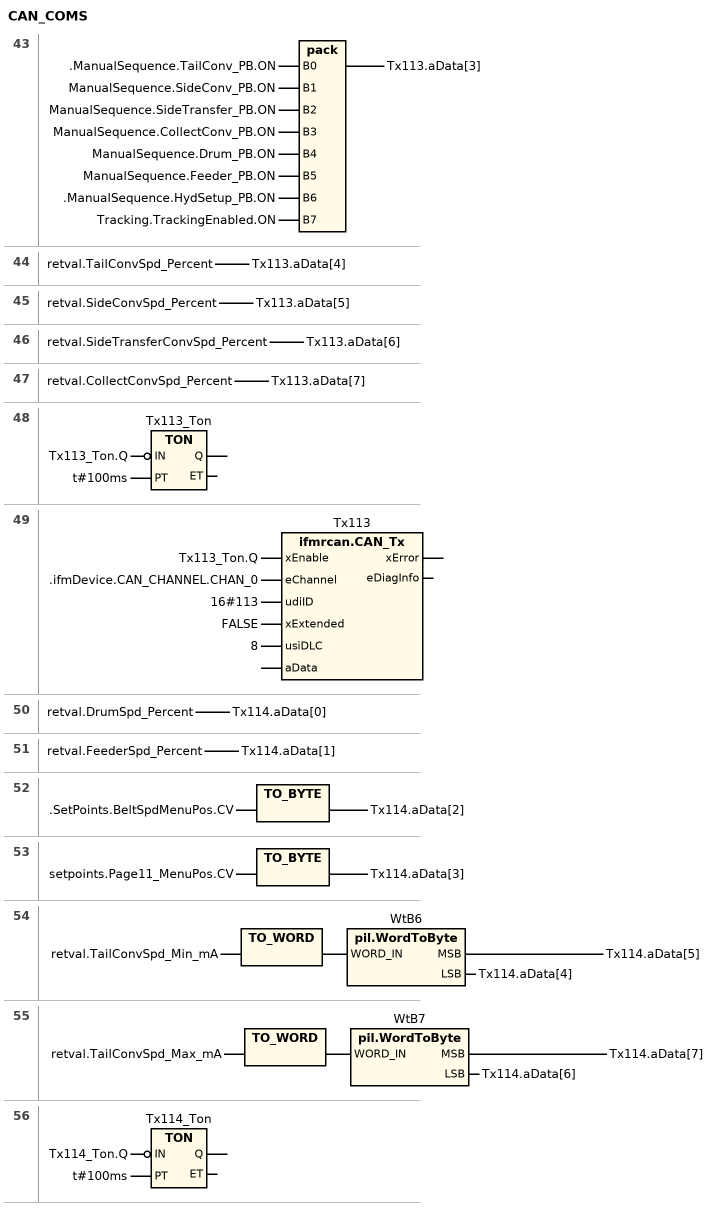
// NETWORK 43
Tx113.aData[3] := pack(B0 := .ManualSequence.TailConv_PB.ON, B1 := ManualSequence.SideConv_PB.ON, B2 := ManualSequence.SideTransfer_PB.ON, B3 := ManualSequence.CollectConv_PB.ON, B4 := ManualSequence.Drum_PB.ON, B5 := ManualSequence.Feeder_PB.ON, B6 := .ManualSequence.HydSetup_PB.ON, B7 := Tracking.TrackingEnabled.ON);

// NETWORK 44
Tx113.aData[4] := retval.TailConvSpd_Percent;

// NETWORK 45
Tx113.aData[5] := retval.SideConvSpd_Percent;

// NETWORK 46
Tx113.aData[6] := retval.SideTransferConvSpd_Percent;

// NETWORK 47
Tx113.aData[7] := retval.CollectConvSpd_Percent;

// NETWORK 48
Tx113_Ton(IN := NOT Tx113_Ton.Q, PT := t#100ms); // TON

// NETWORK 49
Tx113(
    xEnable := Tx113_Ton.Q,
    eChannel := .ifmDevice.CAN_CHANNEL.CHAN_0,
    udiID := 16#113,
    xExtended := FALSE,
    usiDLC := 8); // ifmrcan.CAN_Tx

// NETWORK 50
Tx114.aData[0] := retval.DrumSpd_Percent;

// NETWORK 51
Tx114.aData[1] := retval.FeederSpd_Percent;

// NETWORK 52
Tx114.aData[2] := TO_BYTE(.SetPoints.BeltSpdMenuPos.CV);

// NETWORK 53
Tx114.aData[3] := TO_BYTE(setpoints.Page11_MenuPos.CV);

// NETWORK 54
WtB6(WORD_IN := TO_WORD(retval.TailConvSpd_Min_mA), LSB => Tx114.aData[4]); // pil.WordToByte
Tx114.aData[5] := WtB6.MSB;

// NETWORK 55
WtB7(WORD_IN := TO_WORD(retval.TailConvSpd_Max_mA), LSB => Tx114.aData[6]); // pil.WordToByte
Tx114.aData[7] := WtB7.MSB;

// NETWORK 56
Tx114_Ton(IN := NOT Tx114_Ton.Q, PT := t#100ms); // TON

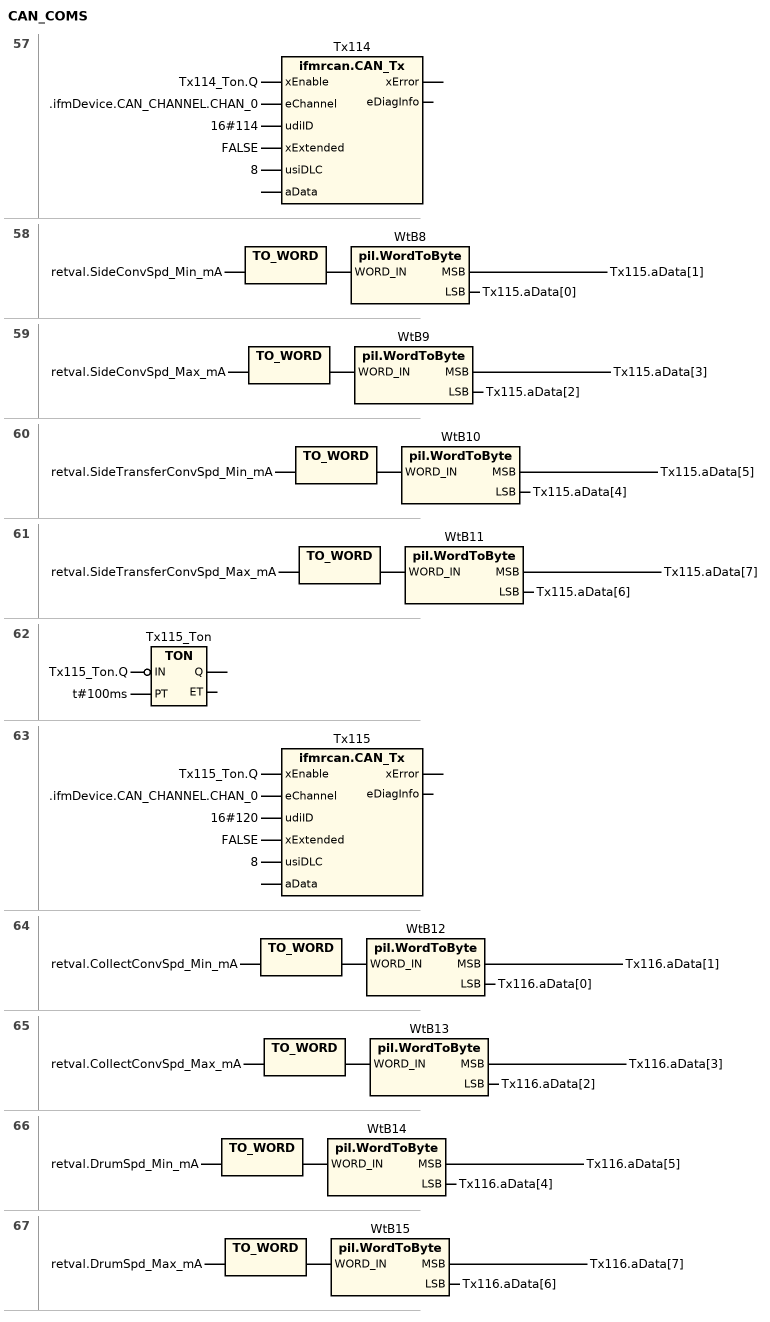
// NETWORK 57
Tx114(
    xEnable := Tx114_Ton.Q,
    eChannel := .ifmDevice.CAN_CHANNEL.CHAN_0,
    udiID := 16#114,
    xExtended := FALSE,
    usiDLC := 8); // ifmrcan.CAN_Tx

// NETWORK 58
WtB8(WORD_IN := TO_WORD(retval.SideConvSpd_Min_mA), LSB => Tx115.aData[0]); // pil.WordToByte
Tx115.aData[1] := WtB8.MSB;

// NETWORK 59
WtB9(WORD_IN := TO_WORD(retval.SideConvSpd_Max_mA), LSB => Tx115.aData[2]); // pil.WordToByte
Tx115.aData[3] := WtB9.MSB;

// NETWORK 60
WtB10(WORD_IN := TO_WORD(retval.SideTransferConvSpd_Min_mA), LSB => Tx115.aData[4]); // pil.WordToByte
Tx115.aData[5] := WtB10.MSB;

// NETWORK 61
WtB11(WORD_IN := TO_WORD(retval.SideTransferConvSpd_Max_mA), LSB => Tx115.aData[6]); // pil.WordToByte
Tx115.aData[7] := WtB11.MSB;

// NETWORK 62
Tx115_Ton(IN := NOT Tx115_Ton.Q, PT := t#100ms); // TON

// NETWORK 63
Tx115(
    xEnable := Tx115_Ton.Q,
    eChannel := .ifmDevice.CAN_CHANNEL.CHAN_0,
    udiID := 16#120,
    xExtended := FALSE,
    usiDLC := 8); // ifmrcan.CAN_Tx

// NETWORK 64
WtB12(WORD_IN := TO_WORD(retval.CollectConvSpd_Min_mA), LSB => Tx116.aData[0]); // pil.WordToByte
Tx116.aData[1] := WtB12.MSB;

// NETWORK 65
WtB13(WORD_IN := TO_WORD(retval.CollectConvSpd_Max_mA), LSB => Tx116.aData[2]); // pil.WordToByte
Tx116.aData[3] := WtB13.MSB;

// NETWORK 66
WtB14(WORD_IN := TO_WORD(retval.DrumSpd_Min_mA), LSB => Tx116.aData[4]); // pil.WordToByte
Tx116.aData[5] := WtB14.MSB;

// NETWORK 67
WtB15(WORD_IN := TO_WORD(retval.DrumSpd_Max_mA), LSB => Tx116.aData[6]); // pil.WordToByte
Tx116.aData[7] := WtB15.MSB;

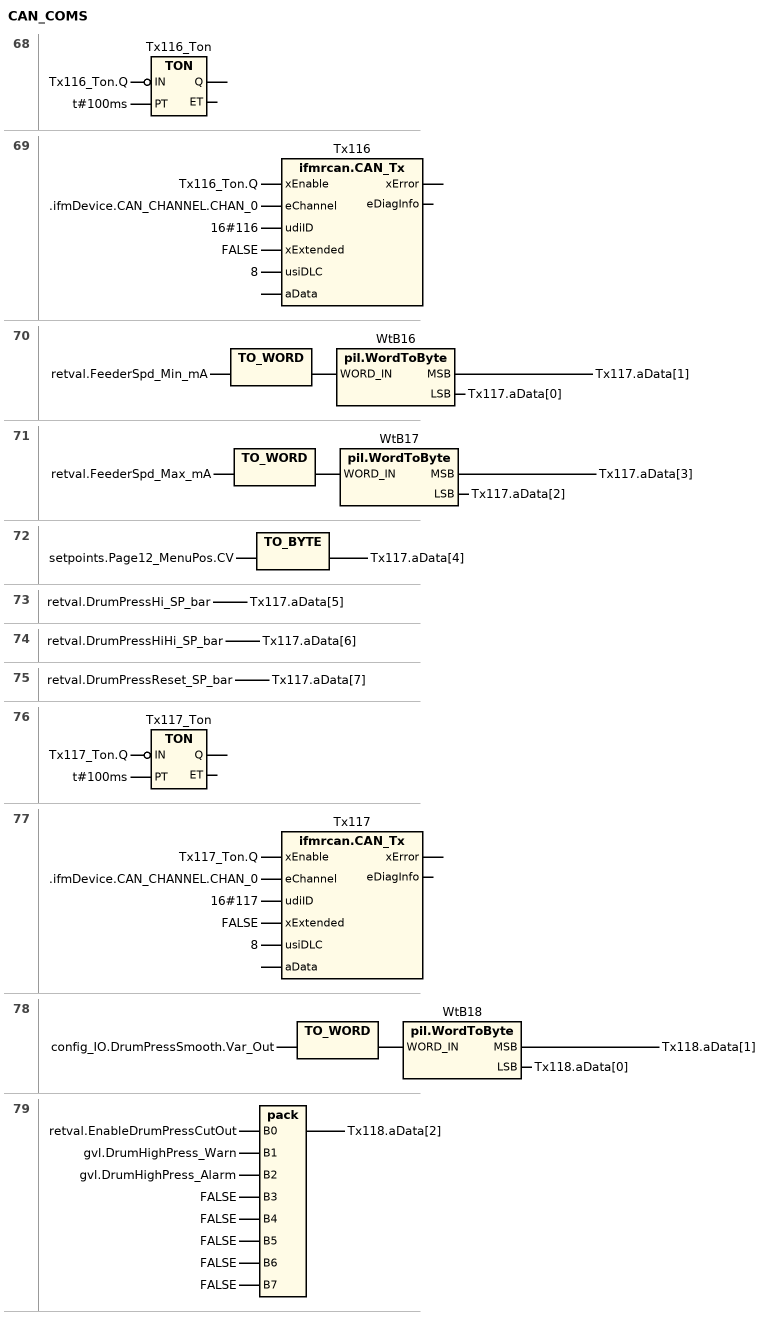
// NETWORK 68
Tx116_Ton(IN := NOT Tx116_Ton.Q, PT := t#100ms); // TON

// NETWORK 69
Tx116(
    xEnable := Tx116_Ton.Q,
    eChannel := .ifmDevice.CAN_CHANNEL.CHAN_0,
    udiID := 16#116,
    xExtended := FALSE,
    usiDLC := 8); // ifmrcan.CAN_Tx

// NETWORK 70
WtB16(WORD_IN := TO_WORD(retval.FeederSpd_Min_mA), LSB => Tx117.aData[0]); // pil.WordToByte
Tx117.aData[1] := WtB16.MSB;

// NETWORK 71
WtB17(WORD_IN := TO_WORD(retval.FeederSpd_Max_mA), LSB => Tx117.aData[2]); // pil.WordToByte
Tx117.aData[3] := WtB17.MSB;

// NETWORK 72
Tx117.aData[4] := TO_BYTE(setpoints.Page12_MenuPos.CV);

// NETWORK 73
Tx117.aData[5] := retval.DrumPressHi_SP_bar;

// NETWORK 74
Tx117.aData[6] := retval.DrumPressHiHi_SP_bar;

// NETWORK 75
Tx117.aData[7] := retval.DrumPressReset_SP_bar;

// NETWORK 76
Tx117_Ton(IN := NOT Tx117_Ton.Q, PT := t#100ms); // TON

// NETWORK 77
Tx117(
    xEnable := Tx117_Ton.Q,
    eChannel := .ifmDevice.CAN_CHANNEL.CHAN_0,
    udiID := 16#117,
    xExtended := FALSE,
    usiDLC := 8); // ifmrcan.CAN_Tx

// NETWORK 78
WtB18(WORD_IN := TO_WORD(config_IO.DrumPressSmooth.Var_Out), LSB => Tx118.aData[0]); // pil.WordToByte
Tx118.aData[1] := WtB18.MSB;

// NETWORK 79
Tx118.aData[2] := pack(B0 := retval.EnableDrumPressCutOut, B1 := gvl.DrumHighPress_Warn, B2 := gvl.DrumHighPress_Alarm, B3 := FALSE, B4 := FALSE, B5 := FALSE, B6 := FALSE, B7 := FALSE);

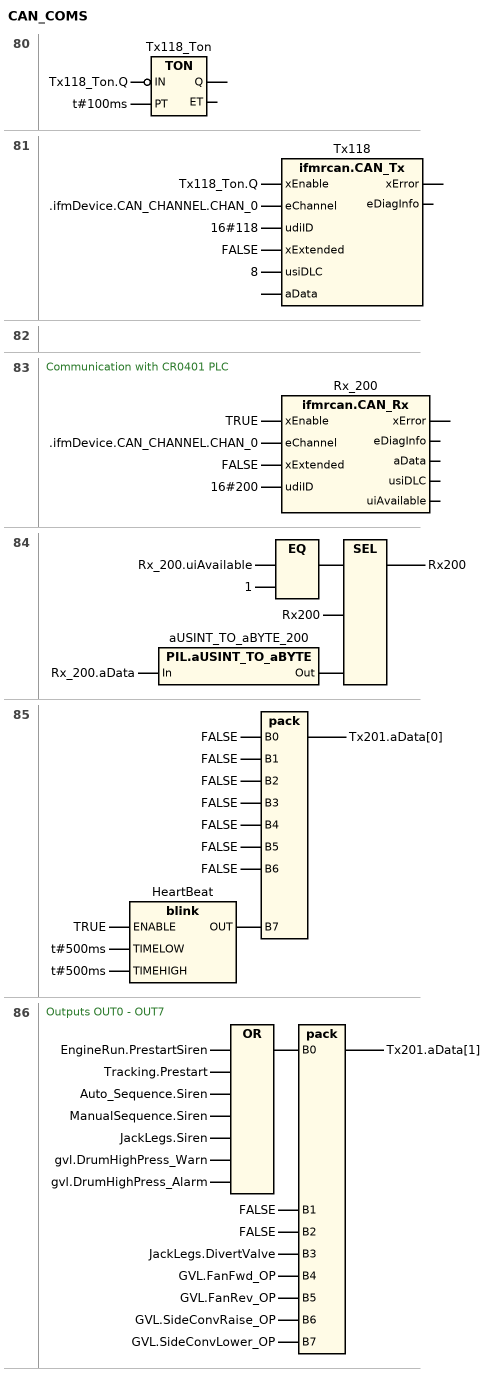
// NETWORK 80
Tx118_Ton(IN := NOT Tx118_Ton.Q, PT := t#100ms); // TON

// NETWORK 81
Tx118(
    xEnable := Tx118_Ton.Q,
    eChannel := .ifmDevice.CAN_CHANNEL.CHAN_0,
    udiID := 16#118,
    xExtended := FALSE,
    usiDLC := 8); // ifmrcan.CAN_Tx

// NETWORK 82

// NETWORK 83
// Communication with CR0401 PLC
Rx_200(xEnable := TRUE, eChannel := .ifmDevice.CAN_CHANNEL.CHAN_0, xExtended := FALSE, udiID := 16#200); // ifmrcan.CAN_Rx

// NETWORK 84
aUSINT_TO_aBYTE_200(In := Rx_200.aData); // PIL.aUSINT_TO_aBYTE
Rx200 := SEL(Rx_200.uiAvailable = 1, Rx200, aUSINT_TO_aBYTE_200.Out);

// NETWORK 85
HeartBeat(ENABLE := TRUE, TIMELOW := t#500ms, TIMEHIGH := t#500ms); // blink
Tx201.aData[0] := pack(B0 := FALSE, B1 := FALSE, B2 := FALSE, B3 := FALSE, B4 := FALSE, B5 := FALSE, B6 := FALSE, B7 := HeartBeat.OUT);

// NETWORK 86
// Outputs OUT0 - OUT7
Tx201.aData[1] := pack(B0 := EngineRun.PrestartSiren OR Tracking.Prestart OR Auto_Sequence.Siren OR ManualSequence.Siren OR JackLegs.Siren OR gvl.DrumHighPress_Warn OR gvl.DrumHighPress_Alarm, B1 := FALSE, B2 := FALSE, B3 := JackLegs.DivertValve, B4 := GVL.FanFwd_OP, B5 := GVL.FanRev_OP, B6 := GVL.SideConvRaise_OP, B7 := GVL.SideConvLower_OP);

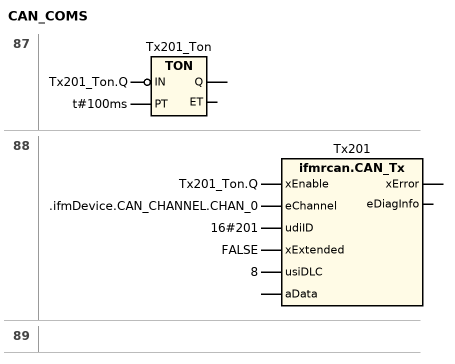
// NETWORK 87
Tx201_Ton(IN := NOT Tx201_Ton.Q, PT := t#100ms); // TON

// NETWORK 88
Tx201(
    xEnable := Tx201_Ton.Q,
    eChannel := .ifmDevice.CAN_CHANNEL.CHAN_0,
    udiID := 16#201,
    xExtended := FALSE,
    usiDLC := 8); // ifmrcan.CAN_Tx

// NETWORK 89

END_PROGRAM

// StandardPLC/Application/Control/ManualSequence
PROGRAM ManualSequence
VAR
	TailConv_PB: pil.PB_Toggle;
	Prestart1: TON;
	ManPrestart1: BOOL;
	Siren: BOOL;
	SideConv_PB: pil.PB_Toggle;
	Prestart2: TON;
	ManPrestart2: BOOL;
	SideTransfer_PB: pil.PB_Toggle;
	Prestart3: TON;
	ManPrestart3: BOOL;
	CollectConv_PB: pil.PB_Toggle;
	Prestart4: TON;
	ManPrestart4: BOOL;
	Drum_PB: pil.PB_Toggle;
	Prestart5: TON;
	ManPrestart5: BOOL;
	Feeder_PB: pil.PB_Toggle;
	Prestart6: TON;
	ManPrestart6: BOOL;
	HydSetup_PB: pil.PB_Toggle;
	Prestart7: TON;
	ManPrestart7: BOOL;
	TailConv_ScaleCurrent: pil.ScaleBlock;
	WaitTon1: ton;
	Flag1: BOOL;
	SideConv_ScaleCurrent: pil.ScaleBlock;
	WaitTon2: ton;
	Flag2: BOOL;
	Flag3: BOOL;
	WaitTon3: ton;
	SideTransfer_ScaleCurrent: pil.ScaleBlock;
	Flag4: BOOL;
	CollectConv_ScaleCurrent: pil.ScaleBlock;
	WaitTon4: ton;
	Flag5: BOOL;
	WaitTon5: ton;
	Drum_ScaleCurrent: pil.ScaleBlock;
	Flag6: BOOL;
	WaitTon6: ton;
	Feeder_ScaleCurrent: pil.ScaleBlock;
	
	// mods to help with the ramp down function for the trommel - stop damage to the valves 2-12-2024
	RAMP_DRUM_SP_OP: UTIL.RAMP_INT;
	RAMP_DRUM_SP_OP_ASCEND: INT:=1000;
	RAMP_DRUM_SP_OP_DESCEND: INT:=100;
	RAMP_DRUM_SP_OP_TIME_BASE: TIME:=T#1S;
	RAMP_DRUM_SP_OP_TIME_RESET: BOOL;
	Flag5_TOF: TOF;
	TestFlag5: BOOL;
END_VAR
VAR // added by the converter: edge detectors and wires of the graphical bodies
    _w1, _w2 : BOOL;
END_VAR

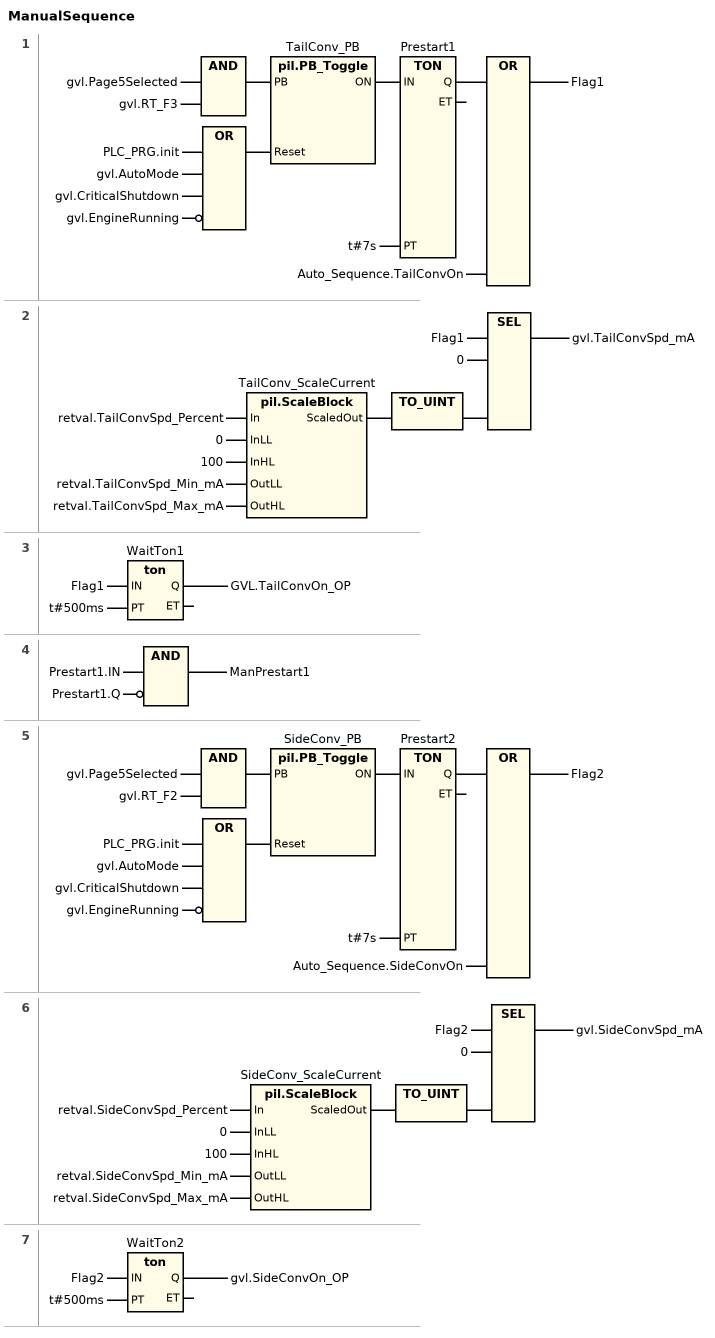
// NETWORK 1
TailConv_PB(PB := gvl.Page5Selected AND gvl.RT_F3, Reset := PLC_PRG.init OR gvl.AutoMode OR gvl.CriticalShutdown OR NOT gvl.EngineRunning); // pil.PB_Toggle
Prestart1(IN := TailConv_PB.ON, PT := t#7s); // TON
Flag1 := Prestart1.Q OR Auto_Sequence.TailConvOn;

// NETWORK 2
TailConv_ScaleCurrent(
    In := retval.TailConvSpd_Percent,
    InLL := 0,
    InHL := 100,
    OutLL := retval.TailConvSpd_Min_mA,
    OutHL := retval.TailConvSpd_Max_mA); // pil.ScaleBlock
gvl.TailConvSpd_mA := SEL(Flag1, 0, TO_UINT(TailConv_ScaleCurrent.ScaledOut));

// NETWORK 3
WaitTon1(IN := Flag1, PT := t#500ms); // ton
GVL.TailConvOn_OP := WaitTon1.Q;

// NETWORK 4
ManPrestart1 := Prestart1.IN AND NOT Prestart1.Q;

// NETWORK 5
SideConv_PB(PB := gvl.Page5Selected AND gvl.RT_F2, Reset := PLC_PRG.init OR gvl.AutoMode OR gvl.CriticalShutdown OR NOT gvl.EngineRunning); // pil.PB_Toggle
Prestart2(IN := SideConv_PB.ON, PT := t#7s); // TON
Flag2 := Prestart2.Q OR Auto_Sequence.SideConvOn;

// NETWORK 6
SideConv_ScaleCurrent(
    In := retval.SideConvSpd_Percent,
    InLL := 0,
    InHL := 100,
    OutLL := retval.SideConvSpd_Min_mA,
    OutHL := retval.SideConvSpd_Max_mA); // pil.ScaleBlock
gvl.SideConvSpd_mA := SEL(Flag2, 0, TO_UINT(SideConv_ScaleCurrent.ScaledOut));

// NETWORK 7
WaitTon2(IN := Flag2, PT := t#500ms); // ton
gvl.SideConvOn_OP := WaitTon2.Q;

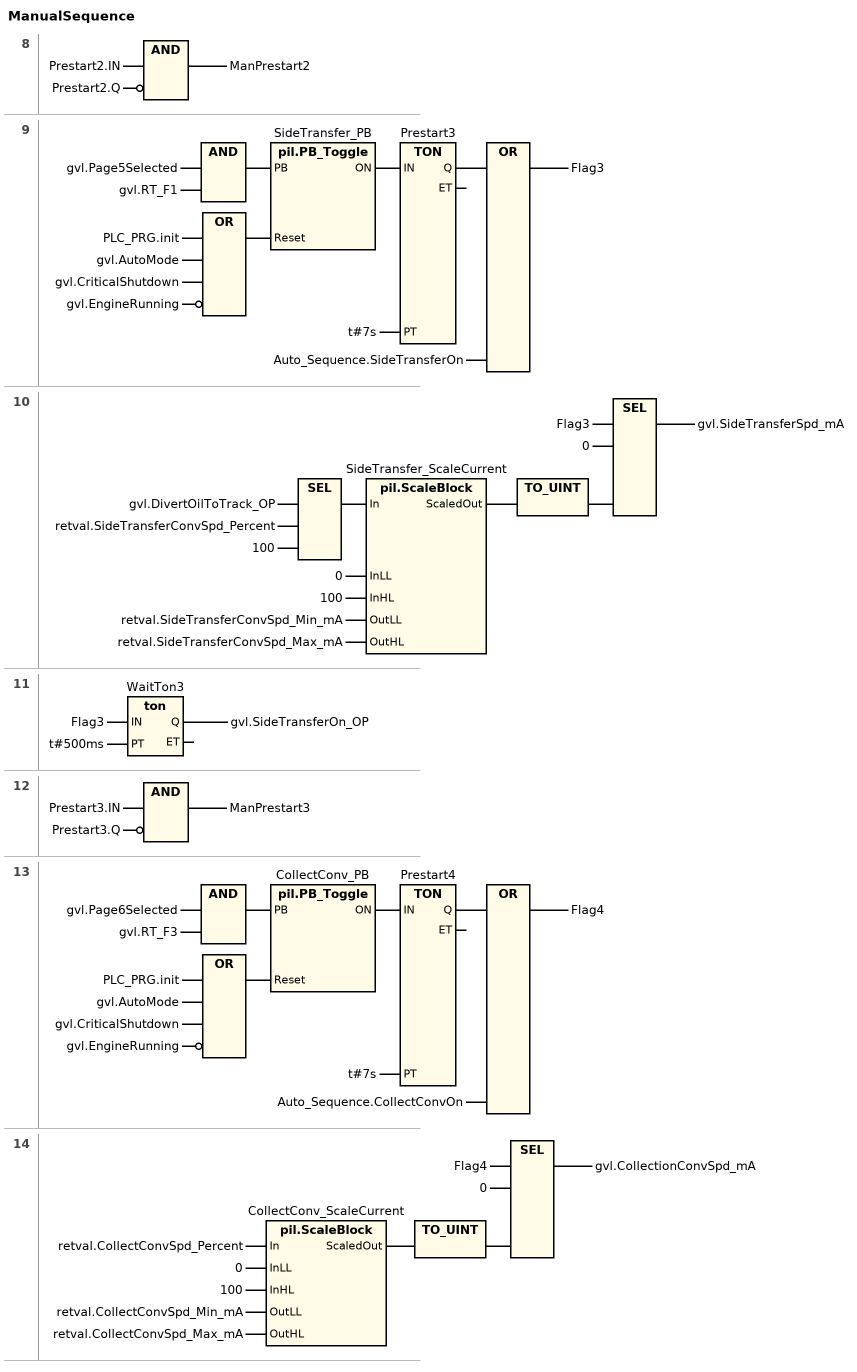
// NETWORK 8
ManPrestart2 := Prestart2.IN AND NOT Prestart2.Q;

// NETWORK 9
SideTransfer_PB(PB := gvl.Page5Selected AND gvl.RT_F1, Reset := PLC_PRG.init OR gvl.AutoMode OR gvl.CriticalShutdown OR NOT gvl.EngineRunning); // pil.PB_Toggle
Prestart3(IN := SideTransfer_PB.ON, PT := t#7s); // TON
Flag3 := Prestart3.Q OR Auto_Sequence.SideTransferOn;

// NETWORK 10
SideTransfer_ScaleCurrent(
    In := SEL(gvl.DivertOilToTrack_OP, retval.SideTransferConvSpd_Percent, 100),
    InLL := 0,
    InHL := 100,
    OutLL := retval.SideTransferConvSpd_Min_mA,
    OutHL := retval.SideTransferConvSpd_Max_mA); // pil.ScaleBlock
gvl.SideTransferSpd_mA := SEL(Flag3, 0, TO_UINT(SideTransfer_ScaleCurrent.ScaledOut));

// NETWORK 11
WaitTon3(IN := Flag3, PT := t#500ms); // ton
gvl.SideTransferOn_OP := WaitTon3.Q;

// NETWORK 12
ManPrestart3 := Prestart3.IN AND NOT Prestart3.Q;

// NETWORK 13
CollectConv_PB(PB := gvl.Page6Selected AND gvl.RT_F3, Reset := PLC_PRG.init OR gvl.AutoMode OR gvl.CriticalShutdown OR NOT gvl.EngineRunning); // pil.PB_Toggle
Prestart4(IN := CollectConv_PB.ON, PT := t#7s); // TON
Flag4 := Prestart4.Q OR Auto_Sequence.CollectConvOn;

// NETWORK 14
CollectConv_ScaleCurrent(
    In := retval.CollectConvSpd_Percent,
    InLL := 0,
    InHL := 100,
    OutLL := retval.CollectConvSpd_Min_mA,
    OutHL := retval.CollectConvSpd_Max_mA); // pil.ScaleBlock
gvl.CollectionConvSpd_mA := SEL(Flag4, 0, TO_UINT(CollectConv_ScaleCurrent.ScaledOut));

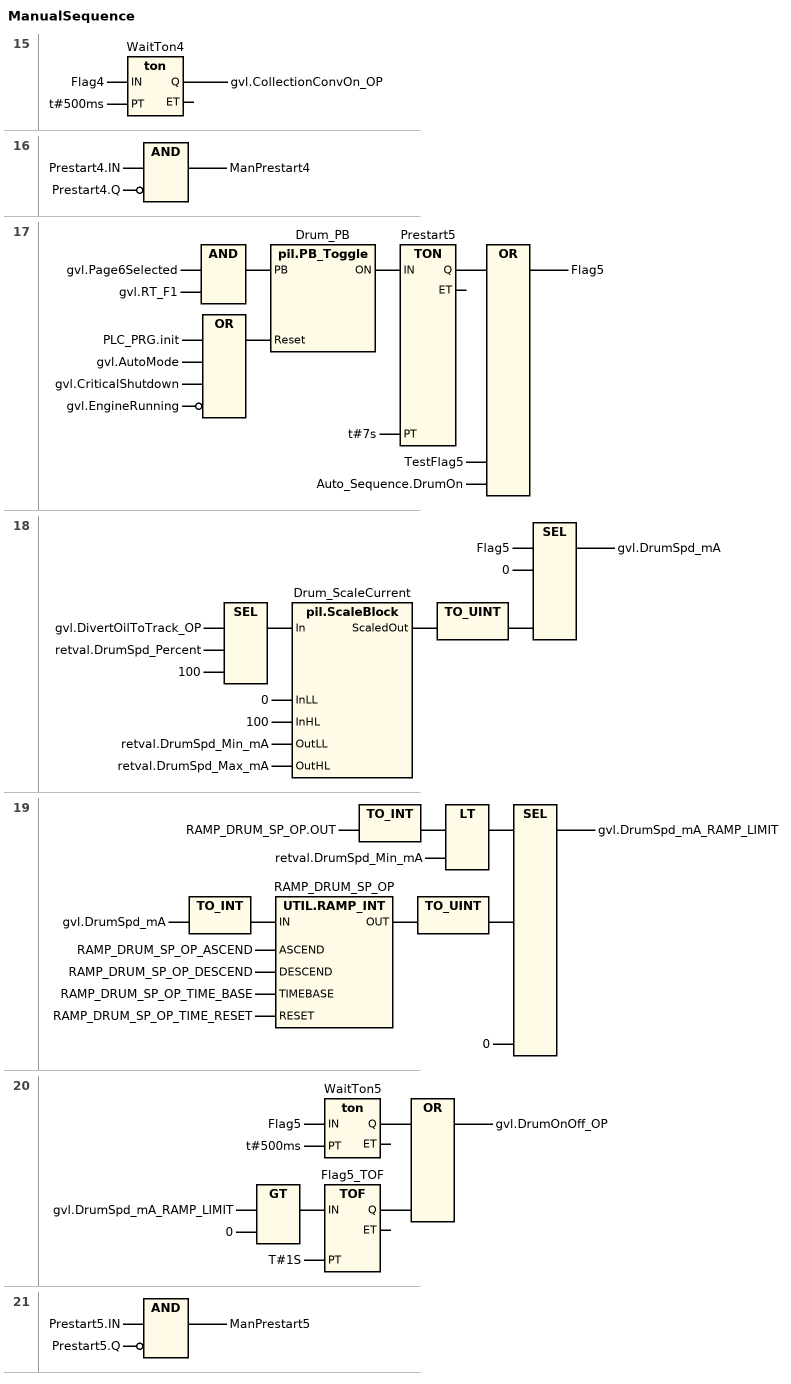
// NETWORK 15
WaitTon4(IN := Flag4, PT := t#500ms); // ton
gvl.CollectionConvOn_OP := WaitTon4.Q;

// NETWORK 16
ManPrestart4 := Prestart4.IN AND NOT Prestart4.Q;

// NETWORK 17
Drum_PB(PB := gvl.Page6Selected AND gvl.RT_F1, Reset := PLC_PRG.init OR gvl.AutoMode OR gvl.CriticalShutdown OR NOT gvl.EngineRunning); // pil.PB_Toggle
Prestart5(IN := Drum_PB.ON, PT := t#7s); // TON
Flag5 := Prestart5.Q OR TestFlag5 OR Auto_Sequence.DrumOn;

// NETWORK 18
Drum_ScaleCurrent(
    In := SEL(gvl.DivertOilToTrack_OP, retval.DrumSpd_Percent, 100),
    InLL := 0,
    InHL := 100,
    OutLL := retval.DrumSpd_Min_mA,
    OutHL := retval.DrumSpd_Max_mA); // pil.ScaleBlock
gvl.DrumSpd_mA := SEL(Flag5, 0, TO_UINT(Drum_ScaleCurrent.ScaledOut));

// NETWORK 19
_w1 := TO_INT(RAMP_DRUM_SP_OP.OUT) < retval.DrumSpd_Min_mA;
RAMP_DRUM_SP_OP(
    IN := TO_INT(gvl.DrumSpd_mA),
    ASCEND := RAMP_DRUM_SP_OP_ASCEND,
    DESCEND := RAMP_DRUM_SP_OP_DESCEND,
    TIMEBASE := RAMP_DRUM_SP_OP_TIME_BASE,
    RESET := RAMP_DRUM_SP_OP_TIME_RESET); // UTIL.RAMP_INT
gvl.DrumSpd_mA_RAMP_LIMIT := SEL(_w1, TO_UINT(RAMP_DRUM_SP_OP.OUT), 0);

// NETWORK 20
WaitTon5(IN := Flag5, PT := t#500ms); // ton
Flag5_TOF(IN := gvl.DrumSpd_mA_RAMP_LIMIT > 0, PT := T#1S); // TOF
gvl.DrumOnOff_OP := WaitTon5.Q OR Flag5_TOF.Q;

// NETWORK 21
ManPrestart5 := Prestart5.IN AND NOT Prestart5.Q;

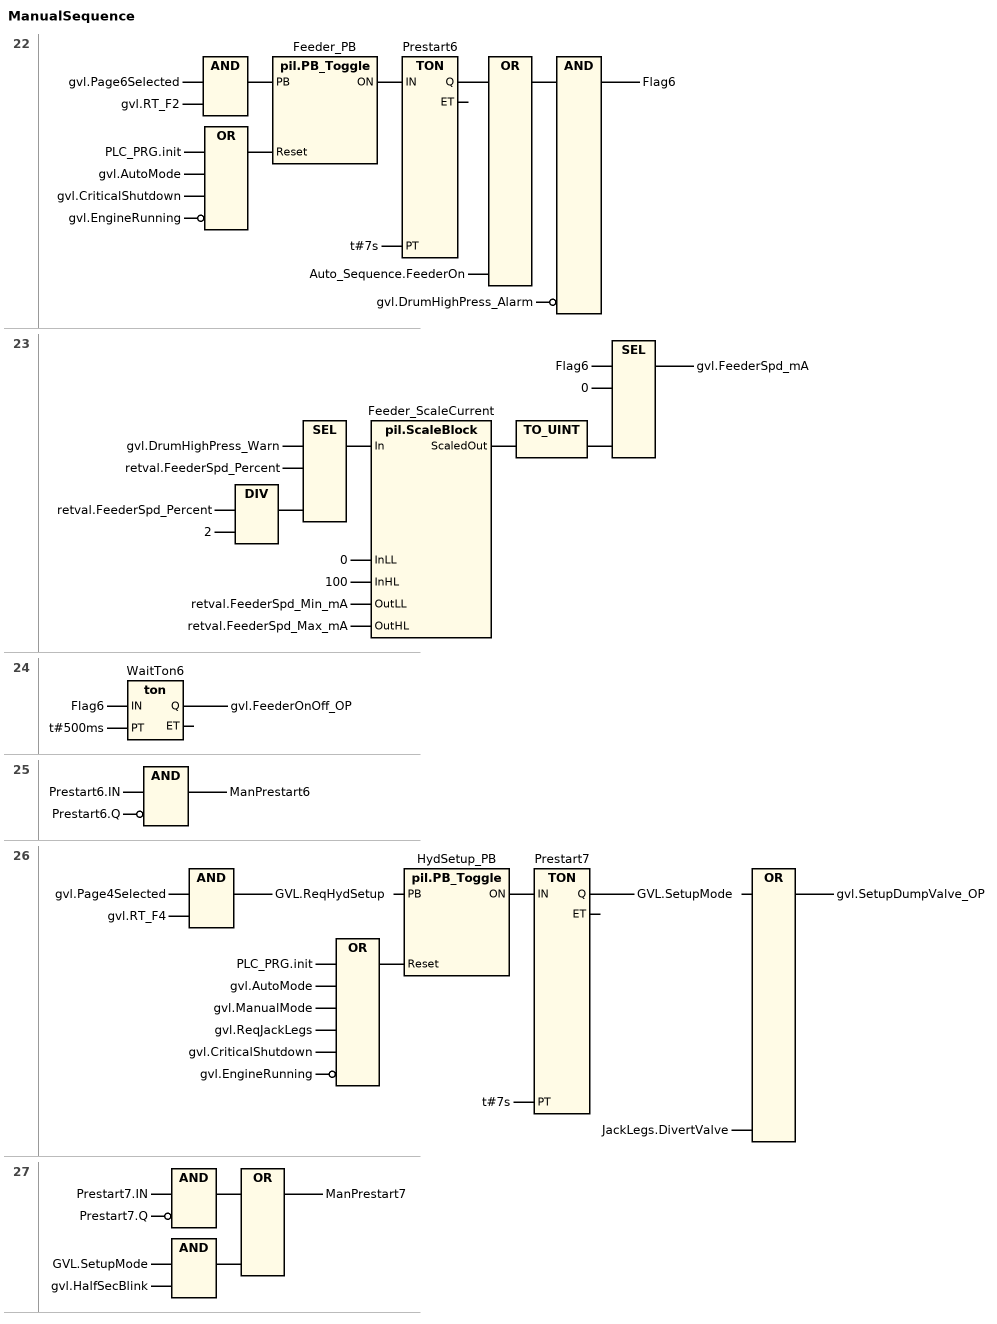
// NETWORK 22
Feeder_PB(PB := gvl.Page6Selected AND gvl.RT_F2, Reset := PLC_PRG.init OR gvl.AutoMode OR gvl.CriticalShutdown OR NOT gvl.EngineRunning); // pil.PB_Toggle
Prestart6(IN := Feeder_PB.ON, PT := t#7s); // TON
Flag6 := (Prestart6.Q OR Auto_Sequence.FeederOn) AND NOT gvl.DrumHighPress_Alarm;

// NETWORK 23
Feeder_ScaleCurrent(
    In := SEL(gvl.DrumHighPress_Warn, retval.FeederSpd_Percent, retval.FeederSpd_Percent / 2),
    InLL := 0,
    InHL := 100,
    OutLL := retval.FeederSpd_Min_mA,
    OutHL := retval.FeederSpd_Max_mA); // pil.ScaleBlock
gvl.FeederSpd_mA := SEL(Flag6, 0, TO_UINT(Feeder_ScaleCurrent.ScaledOut));

// NETWORK 24
WaitTon6(IN := Flag6, PT := t#500ms); // ton
gvl.FeederOnOff_OP := WaitTon6.Q;

// NETWORK 25
ManPrestart6 := Prestart6.IN AND NOT Prestart6.Q;

// NETWORK 26
_w2 := gvl.Page4Selected AND gvl.RT_F4;
GVL.ReqHydSetup := _w2;
HydSetup_PB(PB := _w2, Reset := PLC_PRG.init OR gvl.AutoMode OR gvl.ManualMode OR gvl.ReqJackLegs OR gvl.CriticalShutdown OR NOT gvl.EngineRunning); // pil.PB_Toggle
Prestart7(IN := HydSetup_PB.ON, PT := t#7s); // TON
GVL.SetupMode := Prestart7.Q;
gvl.SetupDumpValve_OP := Prestart7.Q OR JackLegs.DivertValve;

// NETWORK 27
ManPrestart7 := Prestart7.IN AND NOT Prestart7.Q OR GVL.SetupMode AND gvl.HalfSecBlink;

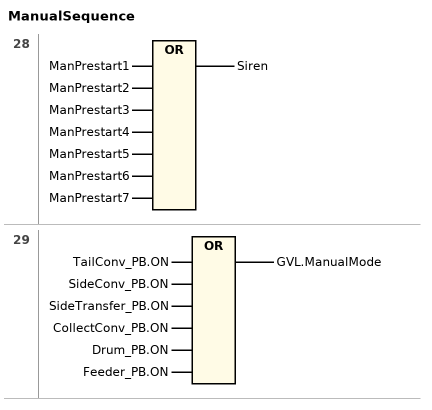
// NETWORK 28
Siren := ManPrestart1 OR ManPrestart2 OR ManPrestart3 OR ManPrestart4 OR ManPrestart5 OR ManPrestart6 OR ManPrestart7;

// NETWORK 29
GVL.ManualMode := TailConv_PB.ON OR SideConv_PB.ON OR SideTransfer_PB.ON OR CollectConv_PB.ON OR Drum_PB.ON OR Feeder_PB.ON;

END_PROGRAM

// StandardPLC/Application/Control/JackLegs
PROGRAM JackLegs
VAR
	JL_SideConv_PB: pil.PB_Toggle;
	Prestart: TON;
	Enable: BOOL;
	Siren: BOOL;
	ResetTon: ton;
	DivertValve: BOOL;
END_VAR
VAR // added by the converter: edge detectors and wires of the graphical bodies
    _w1 : BOOL;
END_VAR

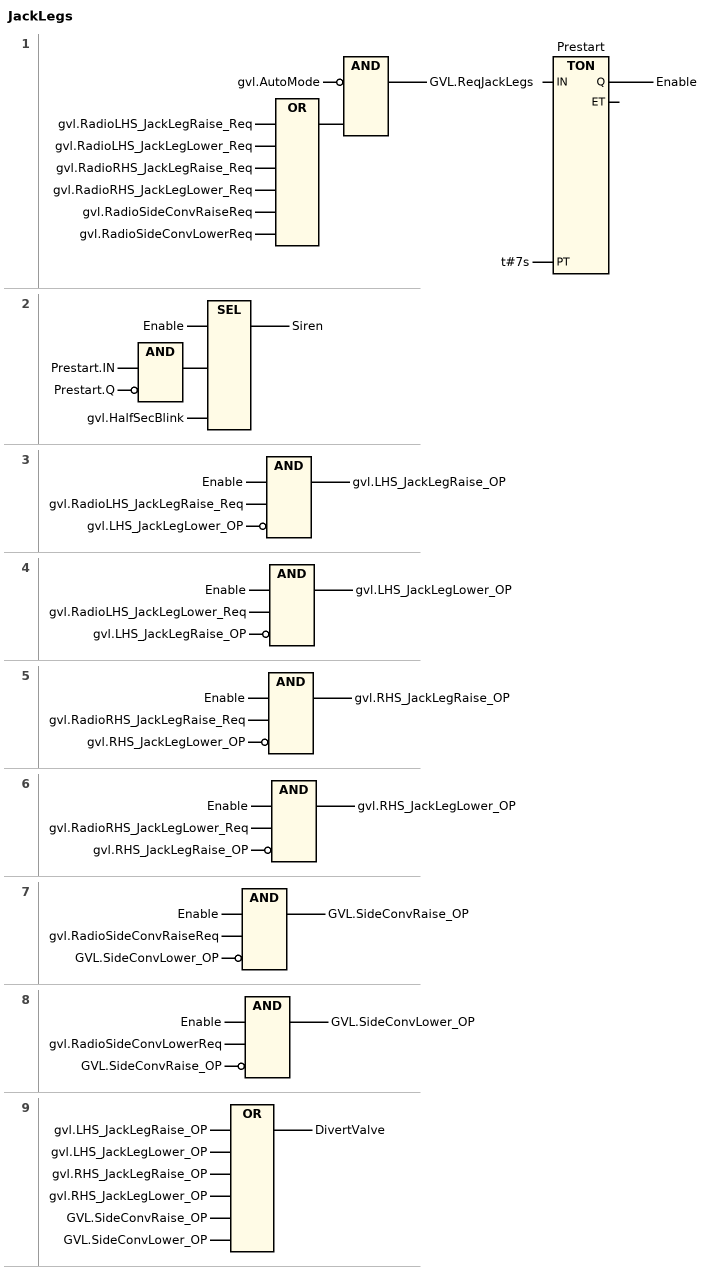
// NETWORK 1
_w1 := NOT gvl.AutoMode AND (gvl.RadioLHS_JackLegRaise_Req OR gvl.RadioLHS_JackLegLower_Req OR gvl.RadioRHS_JackLegRaise_Req OR gvl.RadioRHS_JackLegLower_Req OR gvl.RadioSideConvRaiseReq OR gvl.RadioSideConvLowerReq);
GVL.ReqJackLegs := _w1;
Prestart(IN := _w1, PT := t#7s); // TON
Enable := Prestart.Q;

// NETWORK 2
Siren := SEL(Enable, Prestart.IN AND NOT Prestart.Q, gvl.HalfSecBlink);

// NETWORK 3
gvl.LHS_JackLegRaise_OP := Enable AND gvl.RadioLHS_JackLegRaise_Req AND NOT gvl.LHS_JackLegLower_OP;

// NETWORK 4
gvl.LHS_JackLegLower_OP := Enable AND gvl.RadioLHS_JackLegLower_Req AND NOT gvl.LHS_JackLegRaise_OP;

// NETWORK 5
gvl.RHS_JackLegRaise_OP := Enable AND gvl.RadioRHS_JackLegRaise_Req AND NOT gvl.RHS_JackLegLower_OP;

// NETWORK 6
gvl.RHS_JackLegLower_OP := Enable AND gvl.RadioRHS_JackLegLower_Req AND NOT gvl.RHS_JackLegRaise_OP;

// NETWORK 7
GVL.SideConvRaise_OP := Enable AND gvl.RadioSideConvRaiseReq AND NOT GVL.SideConvLower_OP;

// NETWORK 8
GVL.SideConvLower_OP := Enable AND gvl.RadioSideConvLowerReq AND NOT GVL.SideConvRaise_OP;

// NETWORK 9
DivertValve := gvl.LHS_JackLegRaise_OP OR gvl.LHS_JackLegLower_OP OR gvl.RHS_JackLegRaise_OP OR gvl.RHS_JackLegLower_OP OR GVL.SideConvRaise_OP OR GVL.SideConvLower_OP;

END_PROGRAM

// StandardPLC/Application/Set Points/SetPoints
PROGRAM SetPoints
VAR
	Wait: TON;
	FastBlink: BLINK;
	FastTrig: R_TRIG;
	BeltSpdMenuPos: CTUD;
	TailConvSpd_SP_Count: SP_CountX1;
	SideConvSpd_SP_Count: SP_CountX1;
	SideTransferSpd_SP_Count: SP_CountX1;
	CollectConvSpd_SP_Count: SP_CountX1;
	DrumSpd_SP_Count: SP_CountX1;
	FeederSpd_SP_Count: SP_CountX1;
	Page11_MenuPos: CTUD;
	TailConvSpd_Min_mA_Count: SP_CountX10;
	TailConvSpd_Max_mA_Count: SP_CountX10;
	SideConvSpd_Min_mA_Count: SP_CountX10;
	SideConvSpd_Max_mA_Count: SP_CountX10;
	SideTransferSpd_Max_mA_Count: SP_CountX10;
	SideTransferSpd_Min_mA_Count: SP_CountX10;
	CollectionSpd_Min_mA_Count: SP_CountX10;
	CollectionSpd_Max_mA_Count: SP_CountX10;
	DrumSpd_Min_mA_Count: SP_CountX10;
	DrumSpd_Max_mA_Count: SP_CountX10;
	FeederSpd_Min_mA_Count: SP_CountX10;
	FeederSpd_Max_mA_Count: SP_CountX10;
	Page12_MenuPos: CTUD;
	DrumPress_Hi_SP_Count: SP_CountX1;
	DrumPress_HiHi_SP_Count: SP_CountX1;
	DrumPress_Reset_SP_Count: SP_CountX1;
END_VAR
VAR_INPUT
END_VAR

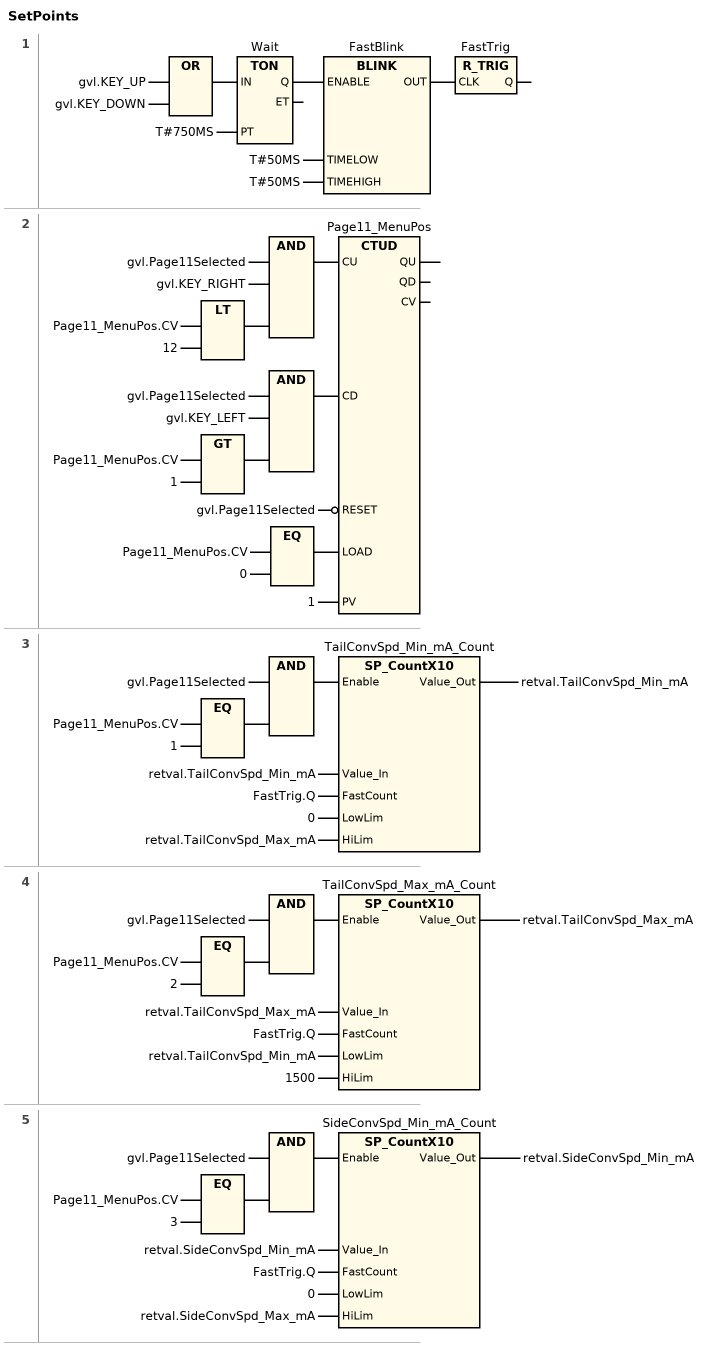
// NETWORK 1
Wait(IN := gvl.KEY_UP OR gvl.KEY_DOWN, PT := T#750MS); // TON
FastBlink(ENABLE := Wait.Q, TIMELOW := T#50MS, TIMEHIGH := T#50MS); // BLINK
FastTrig(CLK := FastBlink.OUT); // R_TRIG

// NETWORK 2
Page11_MenuPos(
    CU := gvl.Page11Selected AND gvl.KEY_RIGHT AND Page11_MenuPos.CV < 12,
    CD := gvl.Page11Selected AND gvl.KEY_LEFT AND Page11_MenuPos.CV > 1,
    RESET := NOT gvl.Page11Selected,
    LOAD := Page11_MenuPos.CV = 0,
    PV := 1); // CTUD

// NETWORK 3
TailConvSpd_Min_mA_Count(
    Enable := gvl.Page11Selected AND Page11_MenuPos.CV = 1,
    Value_In := retval.TailConvSpd_Min_mA,
    FastCount := FastTrig.Q,
    LowLim := 0,
    HiLim := retval.TailConvSpd_Max_mA); // SP_CountX10
retval.TailConvSpd_Min_mA := TailConvSpd_Min_mA_Count.Value_Out;

// NETWORK 4
TailConvSpd_Max_mA_Count(
    Enable := gvl.Page11Selected AND Page11_MenuPos.CV = 2,
    Value_In := retval.TailConvSpd_Max_mA,
    FastCount := FastTrig.Q,
    LowLim := retval.TailConvSpd_Min_mA,
    HiLim := 1500); // SP_CountX10
retval.TailConvSpd_Max_mA := TailConvSpd_Max_mA_Count.Value_Out;

// NETWORK 5
SideConvSpd_Min_mA_Count(
    Enable := gvl.Page11Selected AND Page11_MenuPos.CV = 3,
    Value_In := retval.SideConvSpd_Min_mA,
    FastCount := FastTrig.Q,
    LowLim := 0,
    HiLim := retval.SideConvSpd_Max_mA); // SP_CountX10
retval.SideConvSpd_Min_mA := SideConvSpd_Min_mA_Count.Value_Out;

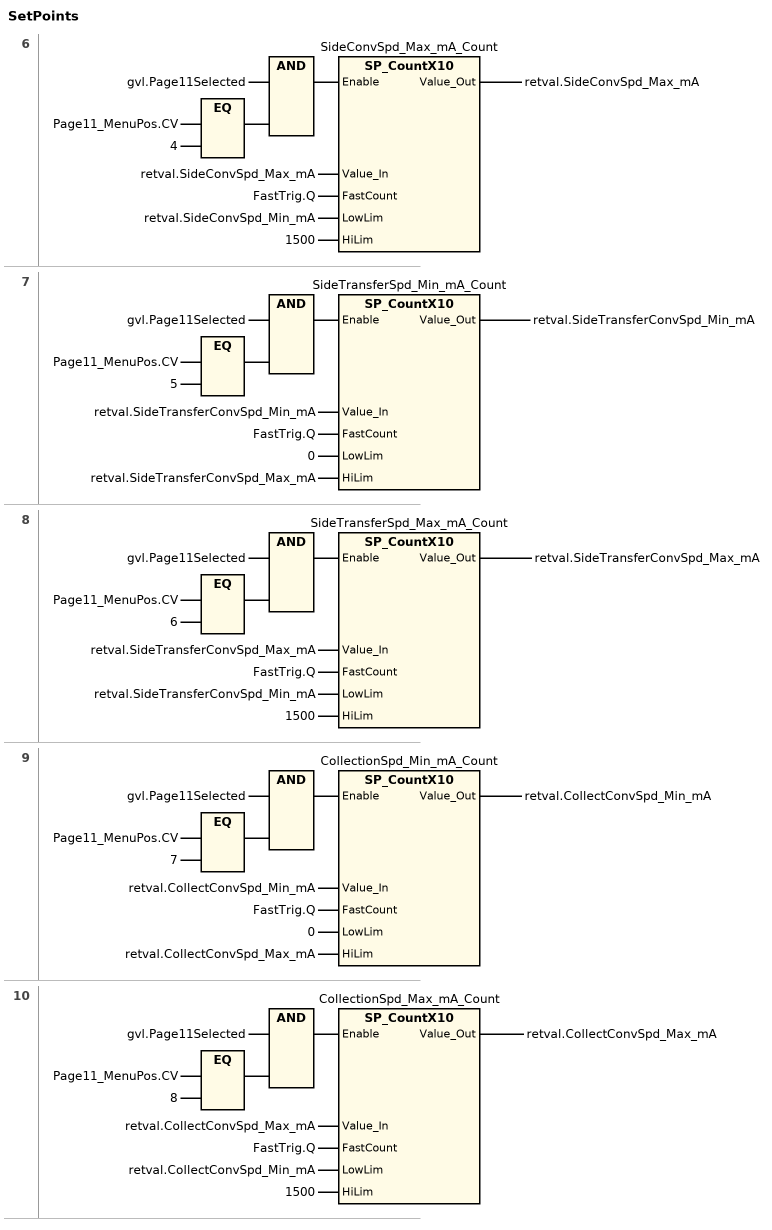
// NETWORK 6
SideConvSpd_Max_mA_Count(
    Enable := gvl.Page11Selected AND Page11_MenuPos.CV = 4,
    Value_In := retval.SideConvSpd_Max_mA,
    FastCount := FastTrig.Q,
    LowLim := retval.SideConvSpd_Min_mA,
    HiLim := 1500); // SP_CountX10
retval.SideConvSpd_Max_mA := SideConvSpd_Max_mA_Count.Value_Out;

// NETWORK 7
SideTransferSpd_Min_mA_Count(
    Enable := gvl.Page11Selected AND Page11_MenuPos.CV = 5,
    Value_In := retval.SideTransferConvSpd_Min_mA,
    FastCount := FastTrig.Q,
    LowLim := 0,
    HiLim := retval.SideTransferConvSpd_Max_mA); // SP_CountX10
retval.SideTransferConvSpd_Min_mA := SideTransferSpd_Min_mA_Count.Value_Out;

// NETWORK 8
SideTransferSpd_Max_mA_Count(
    Enable := gvl.Page11Selected AND Page11_MenuPos.CV = 6,
    Value_In := retval.SideTransferConvSpd_Max_mA,
    FastCount := FastTrig.Q,
    LowLim := retval.SideTransferConvSpd_Min_mA,
    HiLim := 1500); // SP_CountX10
retval.SideTransferConvSpd_Max_mA := SideTransferSpd_Max_mA_Count.Value_Out;

// NETWORK 9
CollectionSpd_Min_mA_Count(
    Enable := gvl.Page11Selected AND Page11_MenuPos.CV = 7,
    Value_In := retval.CollectConvSpd_Min_mA,
    FastCount := FastTrig.Q,
    LowLim := 0,
    HiLim := retval.CollectConvSpd_Max_mA); // SP_CountX10
retval.CollectConvSpd_Min_mA := CollectionSpd_Min_mA_Count.Value_Out;

// NETWORK 10
CollectionSpd_Max_mA_Count(
    Enable := gvl.Page11Selected AND Page11_MenuPos.CV = 8,
    Value_In := retval.CollectConvSpd_Max_mA,
    FastCount := FastTrig.Q,
    LowLim := retval.CollectConvSpd_Min_mA,
    HiLim := 1500); // SP_CountX10
retval.CollectConvSpd_Max_mA := CollectionSpd_Max_mA_Count.Value_Out;

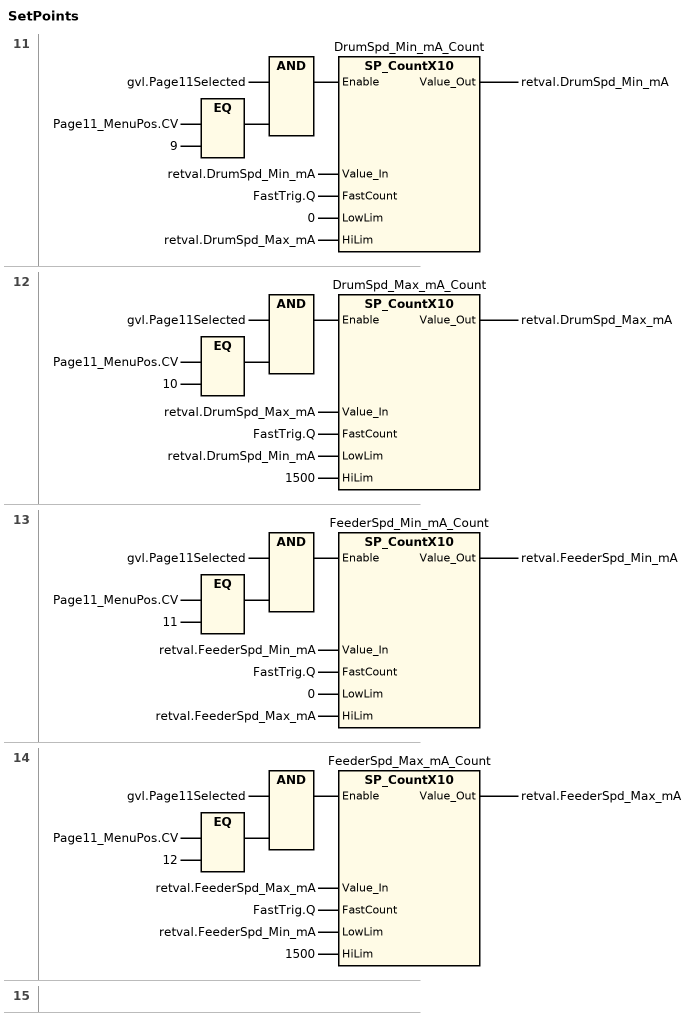
// NETWORK 11
DrumSpd_Min_mA_Count(
    Enable := gvl.Page11Selected AND Page11_MenuPos.CV = 9,
    Value_In := retval.DrumSpd_Min_mA,
    FastCount := FastTrig.Q,
    LowLim := 0,
    HiLim := retval.DrumSpd_Max_mA); // SP_CountX10
retval.DrumSpd_Min_mA := DrumSpd_Min_mA_Count.Value_Out;

// NETWORK 12
DrumSpd_Max_mA_Count(
    Enable := gvl.Page11Selected AND Page11_MenuPos.CV = 10,
    Value_In := retval.DrumSpd_Max_mA,
    FastCount := FastTrig.Q,
    LowLim := retval.DrumSpd_Min_mA,
    HiLim := 1500); // SP_CountX10
retval.DrumSpd_Max_mA := DrumSpd_Max_mA_Count.Value_Out;

// NETWORK 13
FeederSpd_Min_mA_Count(
    Enable := gvl.Page11Selected AND Page11_MenuPos.CV = 11,
    Value_In := retval.FeederSpd_Min_mA,
    FastCount := FastTrig.Q,
    LowLim := 0,
    HiLim := retval.FeederSpd_Max_mA); // SP_CountX10
retval.FeederSpd_Min_mA := FeederSpd_Min_mA_Count.Value_Out;

// NETWORK 14
FeederSpd_Max_mA_Count(
    Enable := gvl.Page11Selected AND Page11_MenuPos.CV = 12,
    Value_In := retval.FeederSpd_Max_mA,
    FastCount := FastTrig.Q,
    LowLim := retval.FeederSpd_Min_mA,
    HiLim := 1500); // SP_CountX10
retval.FeederSpd_Max_mA := FeederSpd_Max_mA_Count.Value_Out;

// NETWORK 15

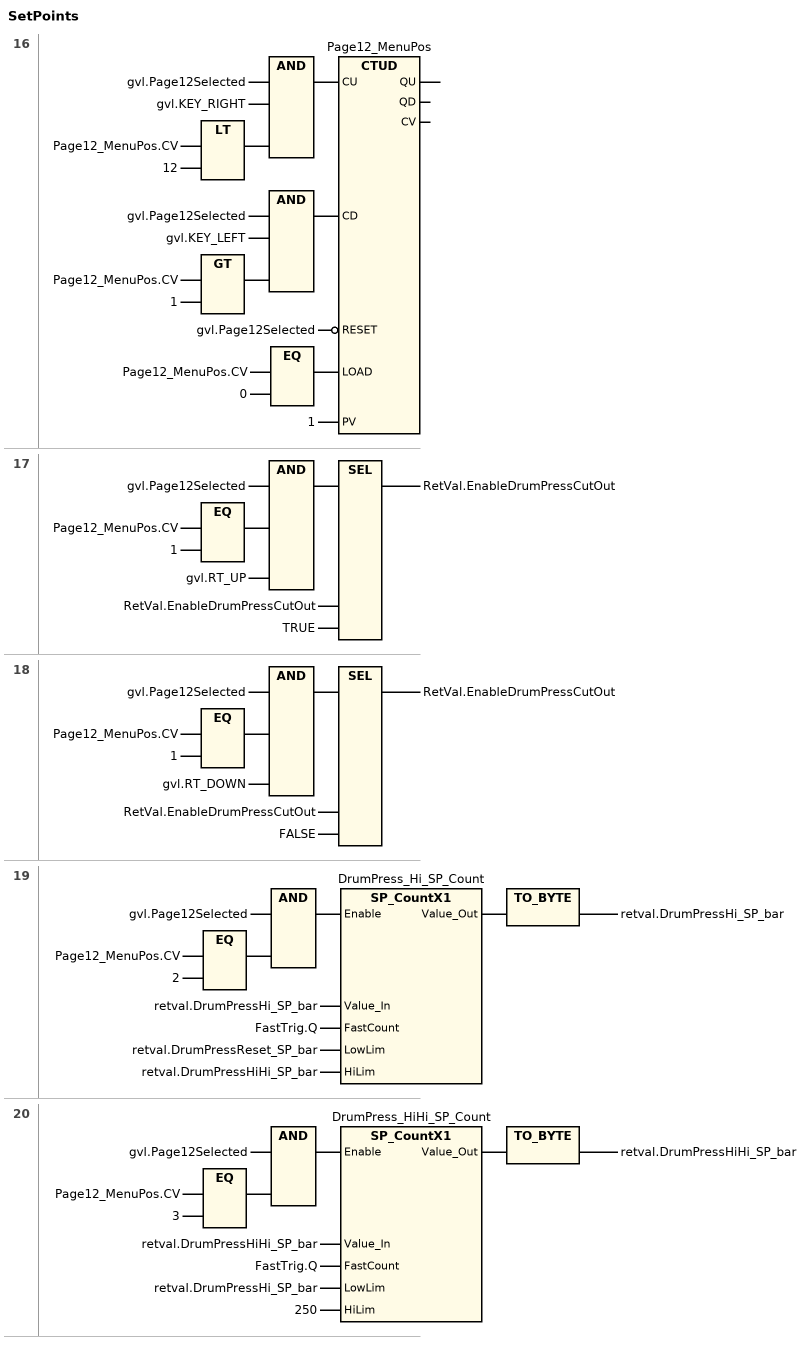
// NETWORK 16
Page12_MenuPos(
    CU := gvl.Page12Selected AND gvl.KEY_RIGHT AND Page12_MenuPos.CV < 12,
    CD := gvl.Page12Selected AND gvl.KEY_LEFT AND Page12_MenuPos.CV > 1,
    RESET := NOT gvl.Page12Selected,
    LOAD := Page12_MenuPos.CV = 0,
    PV := 1); // CTUD

// NETWORK 17
RetVal.EnableDrumPressCutOut := SEL(gvl.Page12Selected AND Page12_MenuPos.CV = 1 AND gvl.RT_UP, RetVal.EnableDrumPressCutOut, TRUE);

// NETWORK 18
RetVal.EnableDrumPressCutOut := SEL(gvl.Page12Selected AND Page12_MenuPos.CV = 1 AND gvl.RT_DOWN, RetVal.EnableDrumPressCutOut, FALSE);

// NETWORK 19
DrumPress_Hi_SP_Count(
    Enable := gvl.Page12Selected AND Page12_MenuPos.CV = 2,
    Value_In := retval.DrumPressHi_SP_bar,
    FastCount := FastTrig.Q,
    LowLim := retval.DrumPressReset_SP_bar,
    HiLim := retval.DrumPressHiHi_SP_bar); // SP_CountX1
retval.DrumPressHi_SP_bar := TO_BYTE(DrumPress_Hi_SP_Count.Value_Out);

// NETWORK 20
DrumPress_HiHi_SP_Count(
    Enable := gvl.Page12Selected AND Page12_MenuPos.CV = 3,
    Value_In := retval.DrumPressHiHi_SP_bar,
    FastCount := FastTrig.Q,
    LowLim := retval.DrumPressHi_SP_bar,
    HiLim := 250); // SP_CountX1
retval.DrumPressHiHi_SP_bar := TO_BYTE(DrumPress_HiHi_SP_Count.Value_Out);

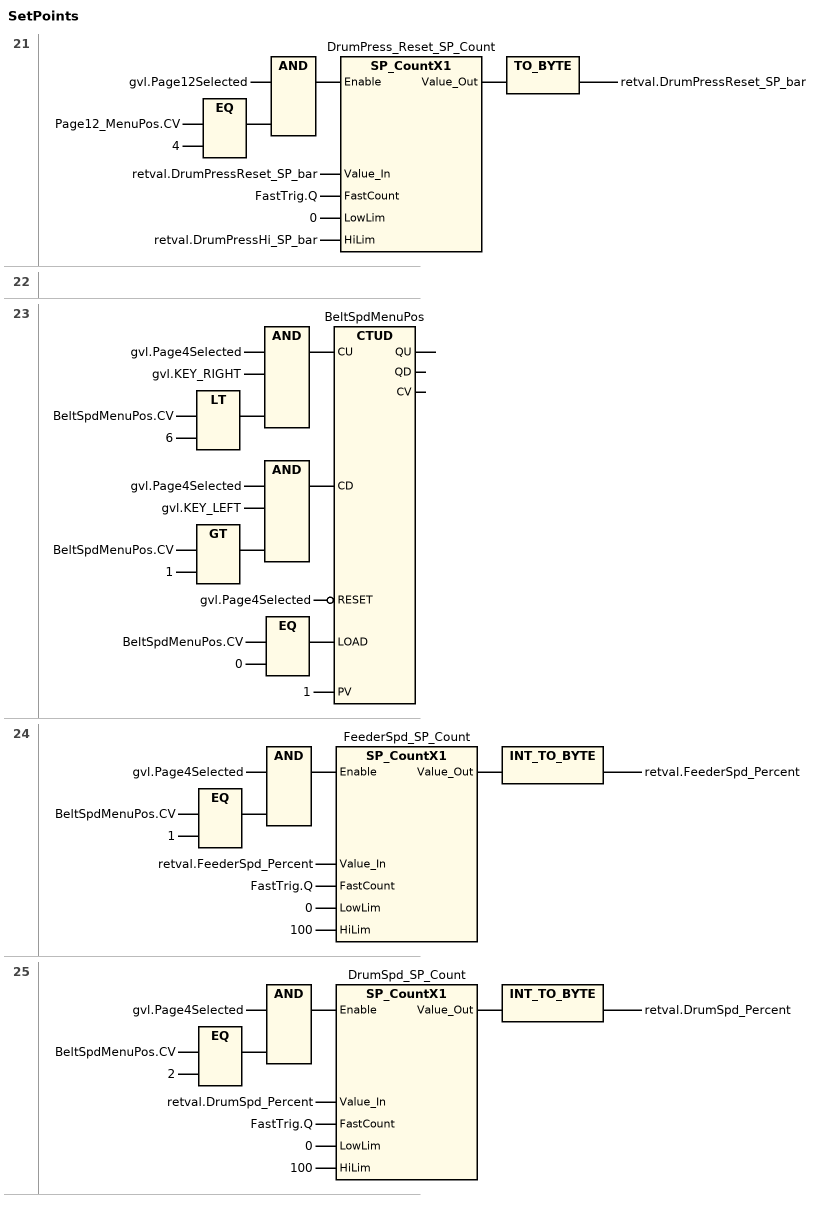
// NETWORK 21
DrumPress_Reset_SP_Count(
    Enable := gvl.Page12Selected AND Page12_MenuPos.CV = 4,
    Value_In := retval.DrumPressReset_SP_bar,
    FastCount := FastTrig.Q,
    LowLim := 0,
    HiLim := retval.DrumPressHi_SP_bar); // SP_CountX1
retval.DrumPressReset_SP_bar := TO_BYTE(DrumPress_Reset_SP_Count.Value_Out);

// NETWORK 22

// NETWORK 23
BeltSpdMenuPos(
    CU := gvl.Page4Selected AND gvl.KEY_RIGHT AND BeltSpdMenuPos.CV < 6,
    CD := gvl.Page4Selected AND gvl.KEY_LEFT AND BeltSpdMenuPos.CV > 1,
    RESET := NOT gvl.Page4Selected,
    LOAD := BeltSpdMenuPos.CV = 0,
    PV := 1); // CTUD

// NETWORK 24
FeederSpd_SP_Count(
    Enable := gvl.Page4Selected AND BeltSpdMenuPos.CV = 1,
    Value_In := retval.FeederSpd_Percent,
    FastCount := FastTrig.Q,
    LowLim := 0,
    HiLim := 100); // SP_CountX1
retval.FeederSpd_Percent := INT_TO_BYTE(FeederSpd_SP_Count.Value_Out);

// NETWORK 25
DrumSpd_SP_Count(
    Enable := gvl.Page4Selected AND BeltSpdMenuPos.CV = 2,
    Value_In := retval.DrumSpd_Percent,
    FastCount := FastTrig.Q,
    LowLim := 0,
    HiLim := 100); // SP_CountX1
retval.DrumSpd_Percent := INT_TO_BYTE(DrumSpd_SP_Count.Value_Out);

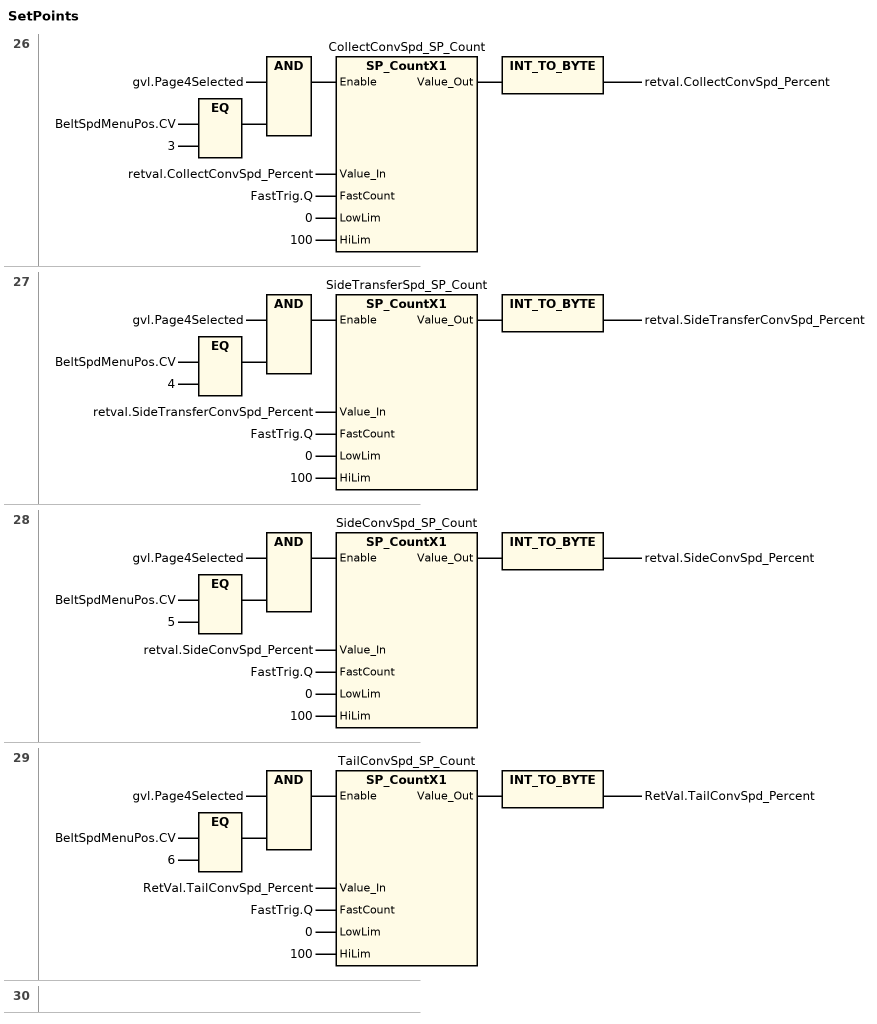
// NETWORK 26
CollectConvSpd_SP_Count(
    Enable := gvl.Page4Selected AND BeltSpdMenuPos.CV = 3,
    Value_In := retval.CollectConvSpd_Percent,
    FastCount := FastTrig.Q,
    LowLim := 0,
    HiLim := 100); // SP_CountX1
retval.CollectConvSpd_Percent := INT_TO_BYTE(CollectConvSpd_SP_Count.Value_Out);

// NETWORK 27
SideTransferSpd_SP_Count(
    Enable := gvl.Page4Selected AND BeltSpdMenuPos.CV = 4,
    Value_In := retval.SideTransferConvSpd_Percent,
    FastCount := FastTrig.Q,
    LowLim := 0,
    HiLim := 100); // SP_CountX1
retval.SideTransferConvSpd_Percent := INT_TO_BYTE(SideTransferSpd_SP_Count.Value_Out);

// NETWORK 28
SideConvSpd_SP_Count(
    Enable := gvl.Page4Selected AND BeltSpdMenuPos.CV = 5,
    Value_In := retval.SideConvSpd_Percent,
    FastCount := FastTrig.Q,
    LowLim := 0,
    HiLim := 100); // SP_CountX1
retval.SideConvSpd_Percent := INT_TO_BYTE(SideConvSpd_SP_Count.Value_Out);

// NETWORK 29
TailConvSpd_SP_Count(
    Enable := gvl.Page4Selected AND BeltSpdMenuPos.CV = 6,
    Value_In := RetVal.TailConvSpd_Percent,
    FastCount := FastTrig.Q,
    LowLim := 0,
    HiLim := 100); // SP_CountX1
RetVal.TailConvSpd_Percent := INT_TO_BYTE(TailConvSpd_SP_Count.Value_Out);

// NETWORK 30

END_PROGRAM

// StandardPLC/Application/Set Points/SP_CountX10
FUNCTION_BLOCK SP_CountX10
VAR_INPUT
	Enable: BOOL;
	Value_In: INT;
	FastCount: BOOL;
	LowLim: INT;
	HiLim: INT;
END_VAR
VAR_OUTPUT
	Value_Out: INT;
END_VAR

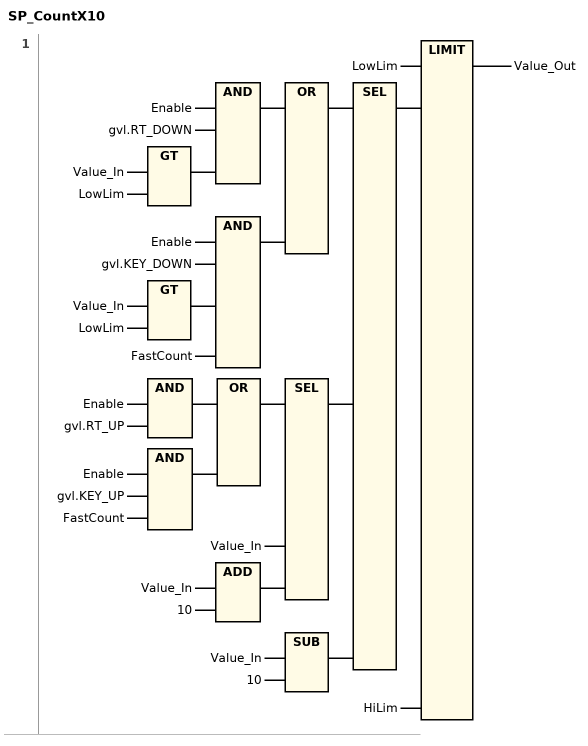
// NETWORK 1
Value_Out := LIMIT(LowLim, SEL(Enable AND gvl.RT_DOWN AND Value_In > LowLim OR Enable AND gvl.KEY_DOWN AND Value_In > LowLim AND FastCount, SEL(Enable AND gvl.RT_UP OR Enable AND gvl.KEY_UP AND FastCount, Value_In, Value_In + 10), Value_In - 10), HiLim);

END_FUNCTION_BLOCK

// StandardPLC/Application/FanCtrl
PROGRAM FanCtrl
VAR
	OneSecTon: TON;
	Step: BYTE;
	WaitTon1: TON;
	WaitTon2: TON;
END_VAR

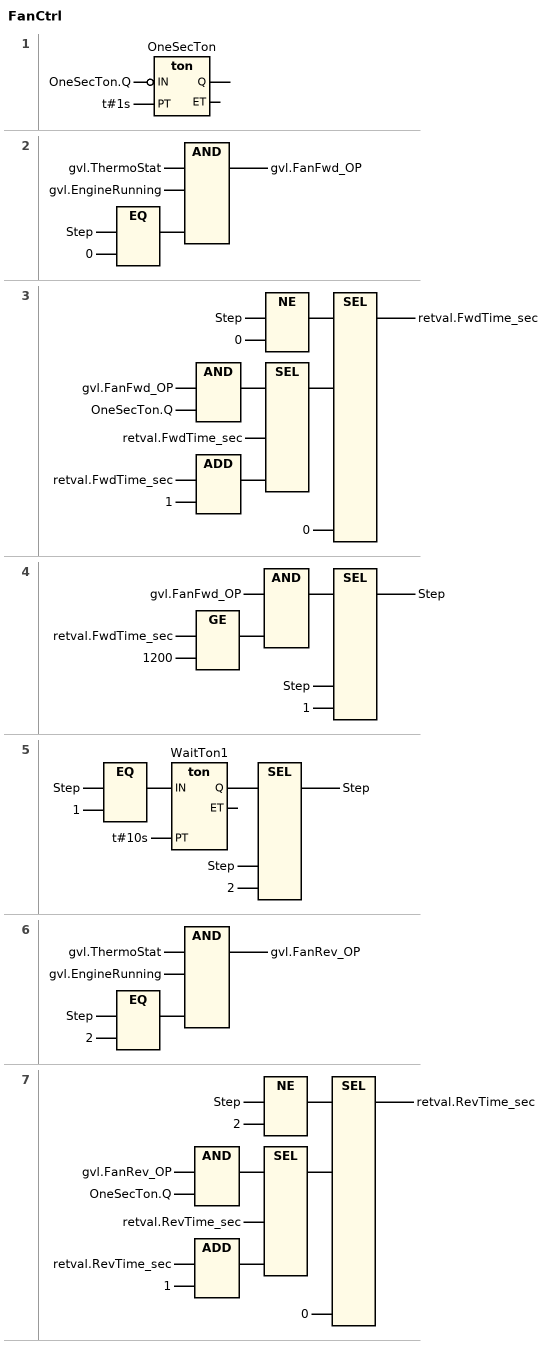
// NETWORK 1
OneSecTon(IN := NOT OneSecTon.Q, PT := t#1s); // ton

// NETWORK 2
gvl.FanFwd_OP := gvl.ThermoStat AND gvl.EngineRunning AND Step = 0;

// NETWORK 3
retval.FwdTime_sec := SEL(Step <> 0, SEL(gvl.FanFwd_OP AND OneSecTon.Q, retval.FwdTime_sec, retval.FwdTime_sec + 1), 0);

// NETWORK 4
Step := SEL(gvl.FanFwd_OP AND retval.FwdTime_sec >= 1200, Step, 1);

// NETWORK 5
WaitTon1(IN := Step = 1, PT := t#10s); // ton
Step := SEL(WaitTon1.Q, Step, 2);

// NETWORK 6
gvl.FanRev_OP := gvl.ThermoStat AND gvl.EngineRunning AND Step = 2;

// NETWORK 7
retval.RevTime_sec := SEL(Step <> 2, SEL(gvl.FanRev_OP AND OneSecTon.Q, retval.RevTime_sec, retval.RevTime_sec + 1), 0);

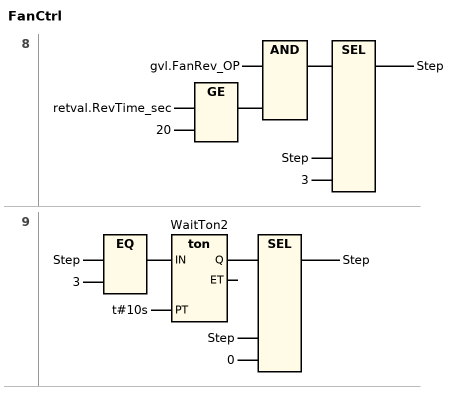
// NETWORK 8
Step := SEL(gvl.FanRev_OP AND retval.RevTime_sec >= 20, Step, 3);

// NETWORK 9
WaitTon2(IN := Step = 3, PT := t#10s); // ton
Step := SEL(WaitTon2.Q, Step, 0);

END_PROGRAM

// StandardPLC/Application/Alarms
PROGRAM Alarms
VAR
	WaitTon1: TON;
	WaitTon2: TON;
	WaitTon3: TON;
	WaitTon4: TON;
	WaitTon5: ton;
	WaitTon6: ton;
	WaitTon7: ton;
	WaitTon8: ton;
END_VAR
VAR // added by the converter: edge detectors and wires of the graphical bodies
    _w1 : BOOL;
END_VAR

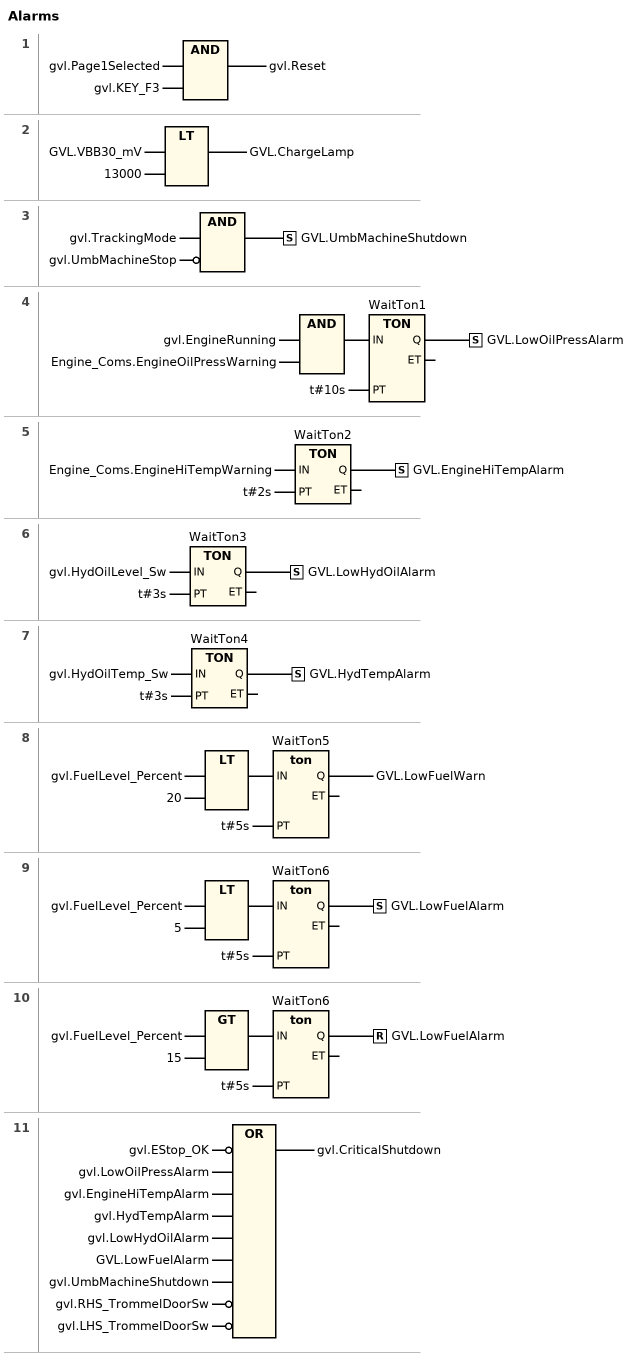
// NETWORK 1
gvl.Reset := gvl.Page1Selected AND gvl.KEY_F3;

// NETWORK 2
GVL.ChargeLamp := GVL.VBB30_mV < 13000;

// NETWORK 3
GVL.UmbMachineShutdown S= gvl.TrackingMode AND NOT gvl.UmbMachineStop;

// NETWORK 4
WaitTon1(IN := gvl.EngineRunning AND Engine_Coms.EngineOilPressWarning, PT := t#10s); // TON
GVL.LowOilPressAlarm S= WaitTon1.Q;

// NETWORK 5
WaitTon2(IN := Engine_Coms.EngineHiTempWarning, PT := t#2s); // TON
GVL.EngineHiTempAlarm S= WaitTon2.Q;

// NETWORK 6
WaitTon3(IN := gvl.HydOilLevel_Sw, PT := t#3s); // TON
GVL.LowHydOilAlarm S= WaitTon3.Q;

// NETWORK 7
WaitTon4(IN := gvl.HydOilTemp_Sw, PT := t#3s); // TON
GVL.HydTempAlarm S= WaitTon4.Q;

// NETWORK 8
WaitTon5(IN := gvl.FuelLevel_Percent < 20, PT := t#5s); // ton
GVL.LowFuelWarn := WaitTon5.Q;

// NETWORK 9
WaitTon6(IN := gvl.FuelLevel_Percent < 5, PT := t#5s); // ton
GVL.LowFuelAlarm S= WaitTon6.Q;

// NETWORK 10
WaitTon6(IN := gvl.FuelLevel_Percent > 15, PT := t#5s); // ton
GVL.LowFuelAlarm R= WaitTon6.Q;

// NETWORK 11
gvl.CriticalShutdown := NOT gvl.EStop_OK OR gvl.LowOilPressAlarm OR gvl.EngineHiTempAlarm OR gvl.HydTempAlarm OR gvl.LowHydOilAlarm OR GVL.LowFuelAlarm OR gvl.UmbMachineShutdown OR NOT gvl.RHS_TrommelDoorSw OR NOT gvl.LHS_TrommelDoorSw;

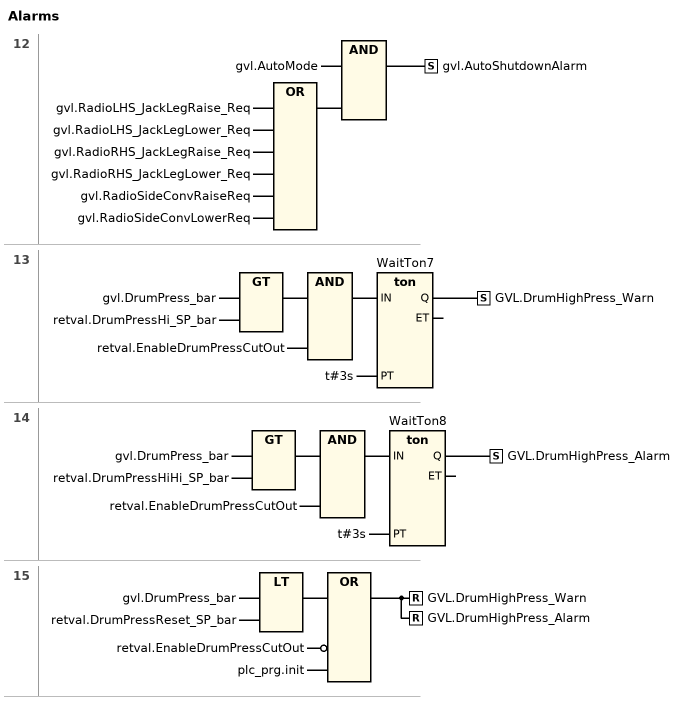
// NETWORK 12
gvl.AutoShutdownAlarm S= gvl.AutoMode AND (gvl.RadioLHS_JackLegRaise_Req OR gvl.RadioLHS_JackLegLower_Req OR gvl.RadioRHS_JackLegRaise_Req OR gvl.RadioRHS_JackLegLower_Req OR gvl.RadioSideConvRaiseReq OR gvl.RadioSideConvLowerReq);

// NETWORK 13
WaitTon7(IN := gvl.DrumPress_bar > retval.DrumPressHi_SP_bar AND retval.EnableDrumPressCutOut, PT := t#3s); // ton
GVL.DrumHighPress_Warn S= WaitTon7.Q;

// NETWORK 14
WaitTon8(IN := gvl.DrumPress_bar > retval.DrumPressHiHi_SP_bar AND retval.EnableDrumPressCutOut, PT := t#3s); // ton
GVL.DrumHighPress_Alarm S= WaitTon8.Q;

// NETWORK 15
_w1 := gvl.DrumPress_bar < retval.DrumPressReset_SP_bar OR NOT retval.EnableDrumPressCutOut OR plc_prg.init;
GVL.DrumHighPress_Warn R= _w1;
GVL.DrumHighPress_Alarm R= _w1;

END_PROGRAM

// Project Information/GetCompany
// This function has been automatically generated from the project information.
{attribute 'signature_flag' := '1073741824'}
{attribute 'register_in_runtime'}
FUNCTION GetCompany : WSTRING
VAR_INPUT
	
END_VAR

GetCompany := "Mtech";

END_FUNCTION

// Project Information/GetTitle
// This function has been automatically generated from the project information.
{attribute 'signature_flag' := '1073741824'}
{attribute 'register_in_runtime'}
FUNCTION GetTitle : WSTRING
VAR_INPUT
	
END_VAR

GetTitle := "T620X PLC";

END_FUNCTION

// Project Information/GetVersion
// This function has been automatically generated from the project information.
{attribute 'signature_flag' := '1073741824'}
{attribute 'register_in_runtime'}
FUNCTION GetVersion : VERSION
VAR_INPUT
	
END_VAR

GetVersion.uiMajor := 1;
GetVersion.uiMinor := 0;
GetVersion.uiServicePack := 3;
GetVersion.uiPatch := 0;

END_FUNCTION

// Project Information/GetTextProperty2
// This function has been automatically generated from the project information.
{attribute 'signature_flag' := '1073741824'}
{attribute 'register_in_runtime'}
FUNCTION GetTextProperty2 : POINTER TO WSTRING
VAR_INPUT
	stKey: WSTRING;
END_VAR

IF stKey = "Company" THEN
	GetTextProperty2 := ADR("Mtech");
ELSIF stKey = "Description" THEN
	GetTextProperty2 := ADR("T620X PLC - pwm ramp mods / sim mods - link fixed for RAMP_LIMIT to the output block");
ELSIF stKey = "Project" THEN
	GetTextProperty2 := ADR("T620X_PLC_CR711S");
ELSIF stKey = "Title" THEN
	GetTextProperty2 := ADR("T620X PLC");
ELSE
	GetTextProperty2 := ADR("");
END_IF

END_FUNCTION

// Project Information/GetNumberProperty
// This function has been automatically generated from the project information.
{attribute 'signature_flag' := '1073741824'}
{attribute 'register_in_runtime'}
FUNCTION GetNumberProperty : DINT
VAR_INPUT
	stKey: WSTRING;
END_VAR

GetNumberProperty := 0;

END_FUNCTION

// Project Information/GetVersionProperty
// This function has been automatically generated from the project information.
{attribute 'signature_flag' := '1073741824'}
{attribute 'register_in_runtime'}
FUNCTION GetVersionProperty : VERSION
VAR_INPUT
	stKey: WSTRING;
END_VAR

IF stKey = "Version" THEN
	GetVersionProperty.uiMajor := 1;
	GetVersionProperty.uiMinor := 0;
	GetVersionProperty.uiServicePack := 3;
	GetVersionProperty.uiPatch := 0;
ELSE
	GetVersionProperty.uiMajor := 0;
	GetVersionProperty.uiMinor := 0;
	GetVersionProperty.uiServicePack := 0;
	GetVersionProperty.uiPatch := 0;
END_IF

END_FUNCTION
